{attribute 'GeneratedUsingTerminal: EL6900-0000-0016'}
{attribute addProperty BoxType "EL6900-0000-0016"}
{attribute addProperty Id "DEVICE_InputsAT %I*DEVICE_Inputs_745C19EA6DEVICE_OutputsAT %Q*DEVICE_Outputs_DAFD38E02WcStateAT %I*WcState_9091E0EB2InfoDataAT %I*InfoData_94A18F5E2"}
{attribute addProperty CRC "1289604254"}
{attribute addProperty Size "12"}
TYPE EL6900_4CDDCC9E EXTENDS EtcSlaveTerminalBase_947E5A46 :
STRUCT
	{attribute addProperty Name "DEVICE_Inputs"}
	DEVICE_Inputs : DEVICE_Inputs_745C19EA;
	{attribute addProperty Name "DEVICE_Outputs"}
	DEVICE_Outputs : DEVICE_Outputs_DAFD38E0;
	{attribute addProperty Name "WcState"}
	WcState : WcState_9091E0EB;
	{attribute addProperty Name "InfoData"}
	InfoData : InfoData_94A18F5E;
END_STRUCT
END_TYPE

(* stored: Version 1.2.0.0, ProductVersion 3.1.4024.9
   DUT EL6900_4CDDCC9E: Id {c6061171-c0a8-412b-8bb5-f5ca517176e6} *)
